{attribute addProperty BoxType "EJ2521-0224-0016"}
{attribute addProperty Id "StatusAT %I*Status_30784993162"}
{attribute addProperty CRC "3116062718"}
{attribute addProperty SizeInBites "16"}
{attribute addProperty SizeInBytes "2"}
TYPE PTO_Status_B9BB57FE :
STRUCT
	{attribute addProperty Name "Status"}
	Status AT %I* : Status_30784993;
END_STRUCT
END_TYPE

(* stored: Version 1.2.0.0, ProductVersion 3.1.4024.9
   DUT PTO_Status_B9BB57FE: Id {305c8ed1-22d8-4247-a945-8f0d7ced7636} *)
